{attribute 'pack_mode' := '1'}
    {attribute 'OPC.UA.DA' := '1'}
    {attribute 'OPC.UA.DA.StructuredType' := '1'}
    (*
    ST_RW_Bool_Memory_HMI_IgnitionExp
    ==================================================
    Generated from Ignition UDT: RW_Bool_Memory
    Total tags: 1
    Generated on: 2025-09-15 13:03:45
    *)
    TYPE ST_RW_Bool_Memory_HMI_IgnitionExp :
    STRUCT
        {attribute 'OPC.UA.DA' := '1'}
        Value : BOOL := FALSE;
    END_STRUCT
    END_TYPE

(* stored: Version 1.1.0.1
   DUT ST_RW_Bool_Memory_HMI_IgnitionExp: Id {b2f6b2ec-b544-4cdf-a1ce-36a4f5ca88c1} *)
